(* Logix 5000 project; controller _2081 vendor 1 type 14 code 77 rev 19.11; software revision 19.01; part 3 of 4 *)
(* tags used below, declared in another part *)
   B10 : DINT[255];   // Product Shift Register
   B23 : DINT[20];   // Fault Bits
   B3 : DINT[10];   // Utility Bits
   B33 : DINT[10];   // Utility Bits
   B36 : DINT[10];   // One-Shots
   B37 : DINT[10];   // Product Location
   C5 : COUNTER[15];   // Line Duration Counters
   F38 : REAL[25];
   i3 : INT;   // Slot 3 16pt DC Input
   i4 : INT;   // Slot 4 16pt DC Input
   IR_1_BITOff : DINT;   // Indirect Addressing BIT Offset
   IR_1_DWOff : DINT;   // Indirect Addressing WORD Offset
   IR_BITOff : DINT;
   IR_DWOff : DINT;
   N26 : DINT[600];   // Write to PLC
   N27 : DINT[400];   // Read from PLC
   N28 : DINT[200];   // Read from PLC
   N32 : DINT[200];
   N32_1 : DINT;   // Recipe to Run Offset Value
   N32_2 : DINT;   // Recipe Copy Utility
   N32_3 : DINT;   // Recipe Copy Utility
   N40 : DINT[256];   // Recipe Shift
   N41 : DINT[256];   // Recipe Shift
   N42 : DINT[256];   // Recipe Shift
   N50 : DINT[2500];   // Stored Recipes
   o2 : INT[8];   // Slot 2 8-pt Analog Output
   Offset : DINT;
   R6 : CONTROL[10];
   S24 : INT;   // Index Register
   T34 : TIMER[30];   // Utility Timers
   T4 : TIMER[32];
(* BGK_OVEN, continued *)

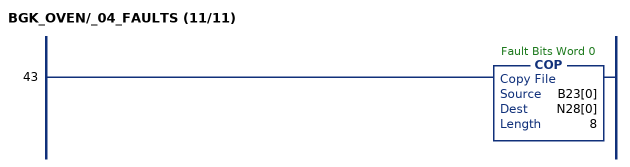
   [picture p24: BGK_OVEN/_04_FAULTS rungs 43-43]
   43: COP(B23[0],N28[0],8);
END_ROUTINE

ROUTINE _05_OIT_MAP   (* ladder *)
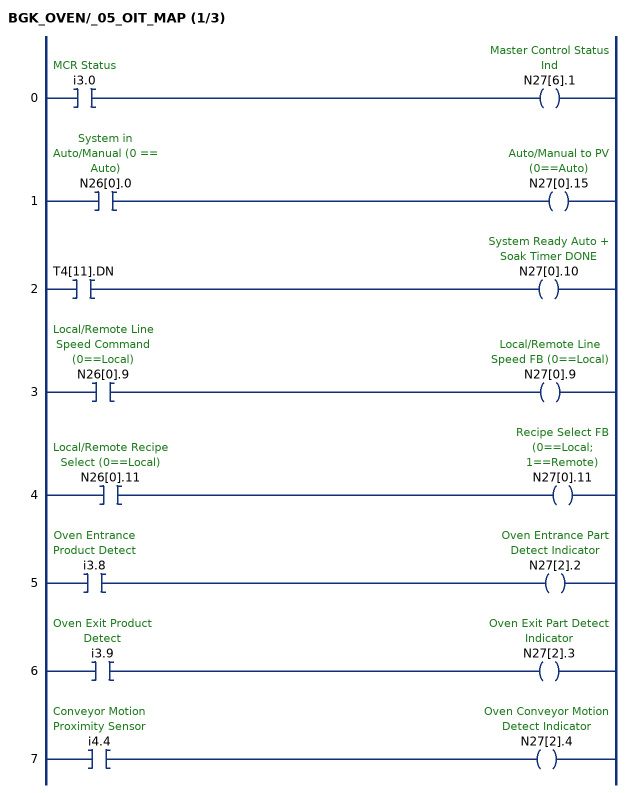
   0: XIC(i3.0)OTE(N27[6].1);
   1: XIC(N26[0].0)OTE(N27[0].15);
   2: XIC(T4[11].DN)OTE(N27[0].10);
   3: XIC(N26[0].9)OTE(N27[0].9);
   4: XIC(N26[0].11)OTE(N27[0].11);
   5: XIC(i3.8)OTE(N27[2].2);
   6: XIC(i3.9)OTE(N27[2].3);
   7: XIC(i4.4)OTE(N27[2].4);
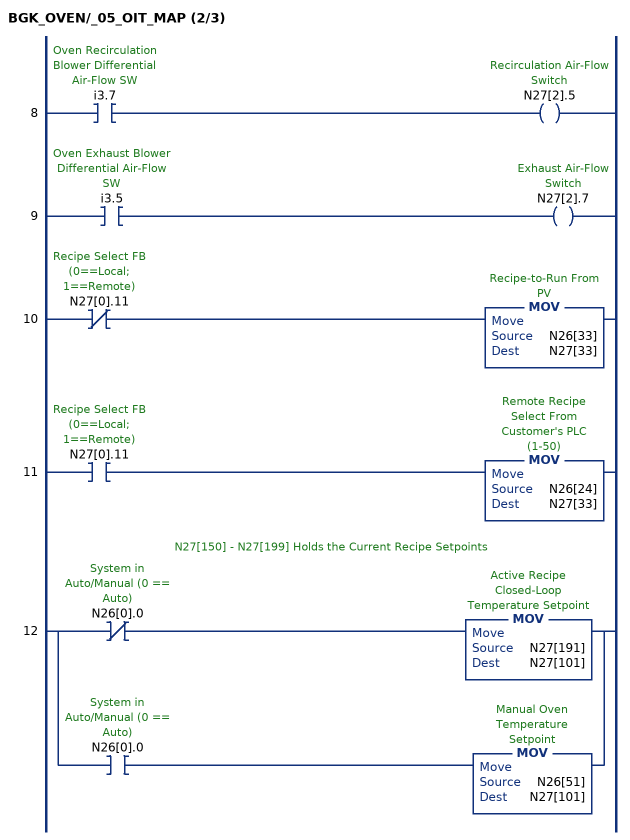
   8: XIC(i3.7)OTE(N27[2].5);
   9: XIC(i3.5)OTE(N27[2].7);
   10: XIO(N27[0].11)MOV(N26[33],N27[33]);
   11: XIC(N27[0].11)MOV(N26[24],N27[33]);
   // N27[150] - N27[199] Holds the Current Recipe Setpoints
   12: [XIO(N26[0].0) MOV(N27[191],N27[101]) ,XIC(N26[0].0) MOV(N26[51],N27[101]) ];
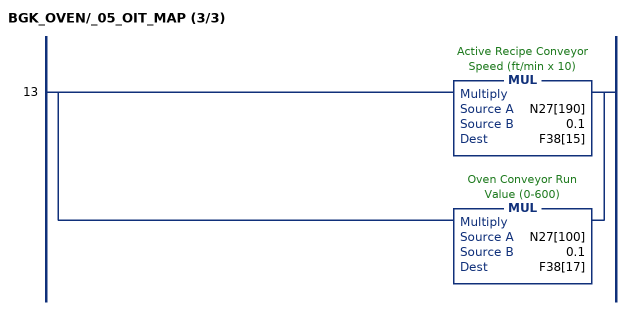
   13: [MUL(N27[190],0.1,F38[15]) ,MUL(N27[100],0.1,F38[17]) ];
END_ROUTINE

ROUTINE _06_SHIFT_REG   (* ladder *)
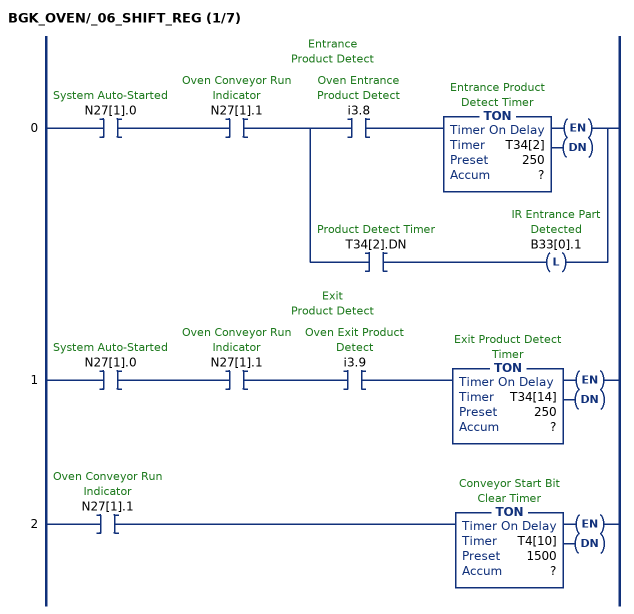
   // Entrance
   // Product Detect
   0: XIC(N27[1].0)XIC(N27[1].1)[XIC(i3.8) TON(T34[2],?,?) ,XIC(T34[2].DN) OTL(B33[0].1) ];
   // Exit
   // Product Detect
   1: XIC(N27[1].0)XIC(N27[1].1)XIC(i3.9)TON(T34[14],?,?);
   2: XIC(N27[1].1)TON(T4[10],?,?);
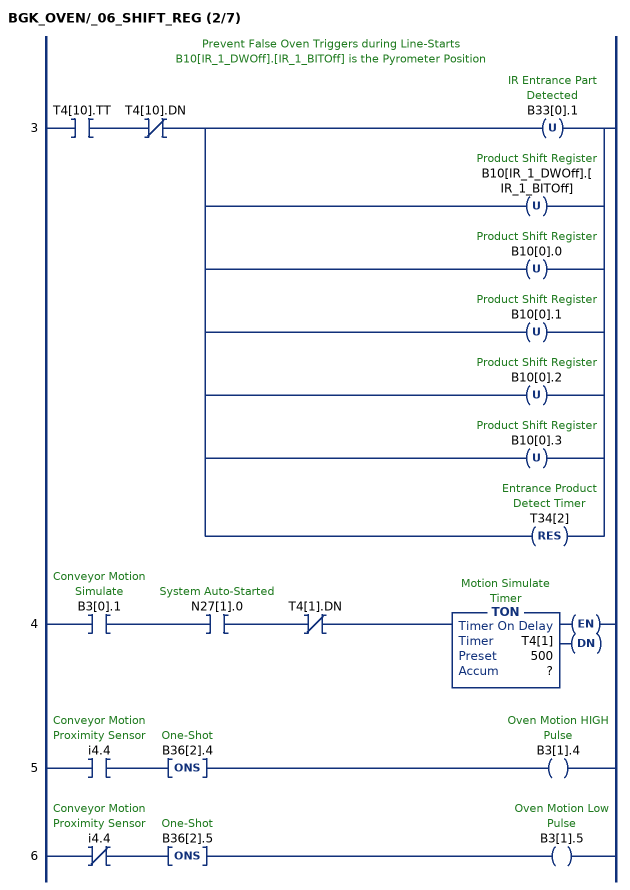
   // Prevent False Oven Triggers during Line-Starts
   // B10[IR_1_DWOff].[IR_1_BITOff] is the Pyrometer Position
   3: XIC(T4[10].TT)XIO(T4[10].DN)[OTU(B33[0].1) ,OTU(B10[IR_1_DWOff].[IR_1_BITOff]) ,OTU(B10[0].0) ,OTU(B10[0].1) ,OTU(B10[0].2) ,OTU(B10[0].3) ,RES(T34[2]) ];
   4: XIC(B3[0].1)XIC(N27[1].0)XIO(T4[1].DN)TON(T4[1],?,?);
   5: XIC(i4.4)ONS(B36[2].4)OTE(B3[1].4);
   6: XIO(i4.4)ONS(B36[2].5)OTE(B3[1].5);
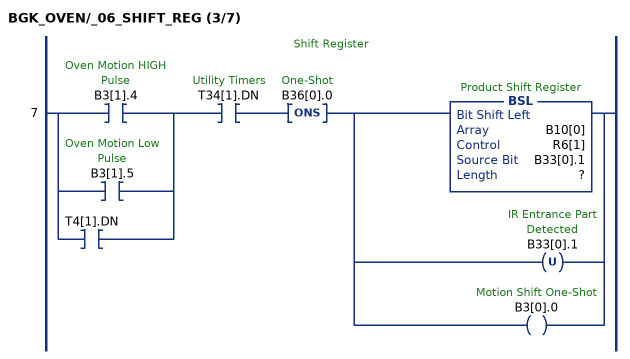
   // Shift Register
   7: [XIC(B3[1].4) ,XIC(B3[1].5) ,XIC(T4[1].DN) ]XIC(T34[1].DN)ONS(B36[0].0)[BSL(B10[0],R6[1],B33[0].1,?) ,OTU(B33[0].1) ,OTE(B3[0].0) ];
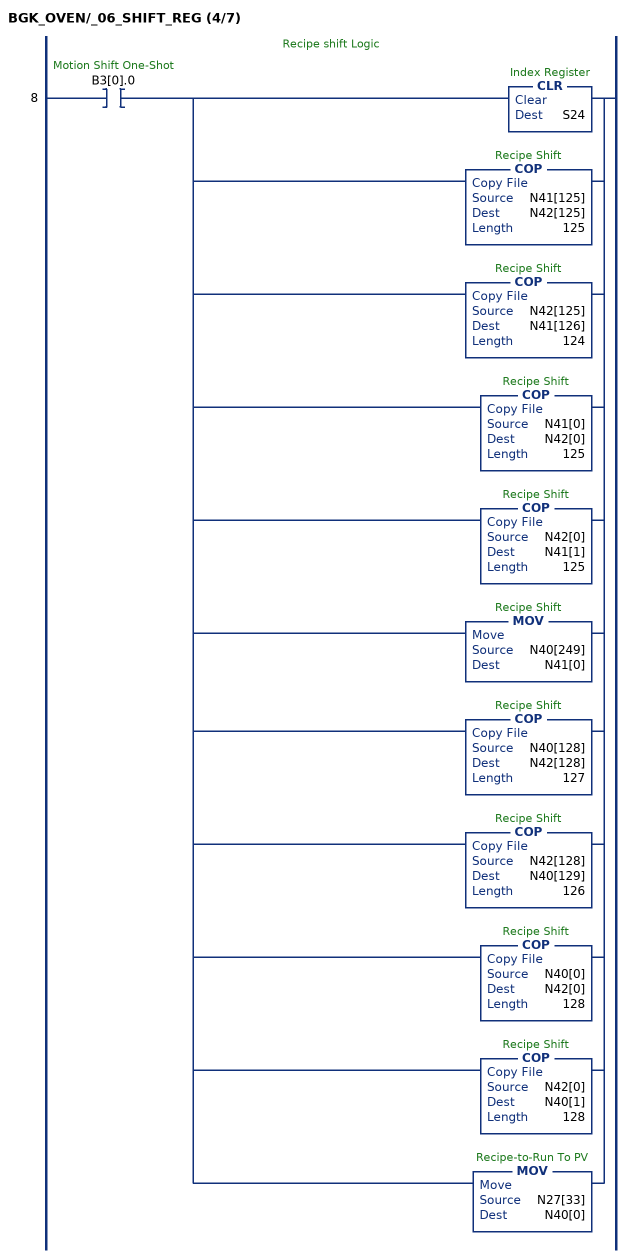
   // Recipe shift Logic
   8: XIC(B3[0].0)[CLR(S24) ,COP(N41[125],N42[125],125) ,COP(N42[125],N41[126],124) ,COP(N41[0],N42[0],125) ,COP(N42[0],N41[1],125) ,MOV(N40[249],N41[0]) ,COP(N40[128],N42[128],127) ,COP(N42[128],N40[129],126) ,COP(N40[0],N42[0],128) ,COP(N42[0],N40[1],128) ,MOV(N27[33],N40[0]) ];
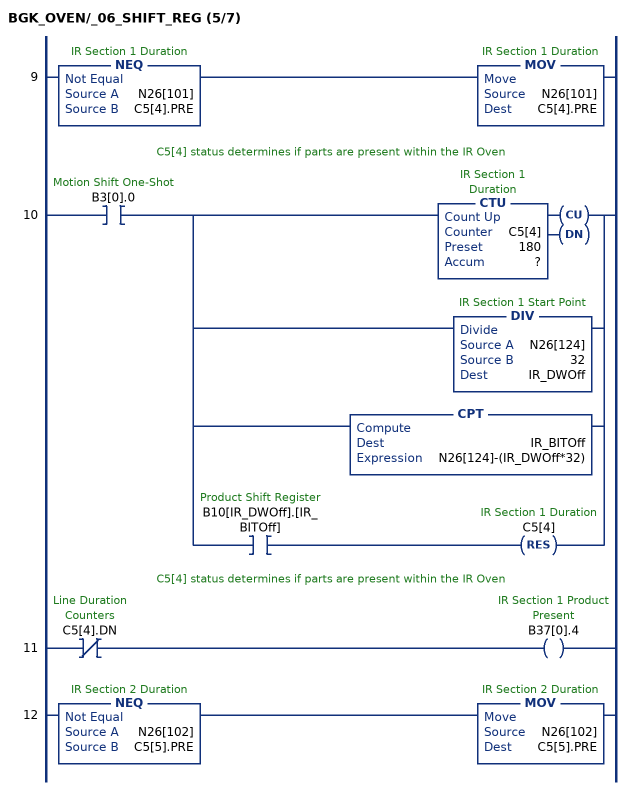
   9: NEQ(N26[101],C5[4].PRE)MOV(N26[101],C5[4].PRE);
   // C5[4] status determines if parts are present within the IR Oven
   10: XIC(B3[0].0)[CTU(C5[4],?,?) ,[DIV(N26[124],32,IR_DWOff) ,CPT(IR_BITOff,N26[124]-(IR_DWOff*32)) ] ,XIC(B10[IR_DWOff].[IR_BITOff]) RES(C5[4]) ];
   // C5[4] status determines if parts are present within the IR Oven
   11: XIO(C5[4].DN)OTE(B37[0].4);
   12: NEQ(N26[102],C5[5].PRE)MOV(N26[102],C5[5].PRE);
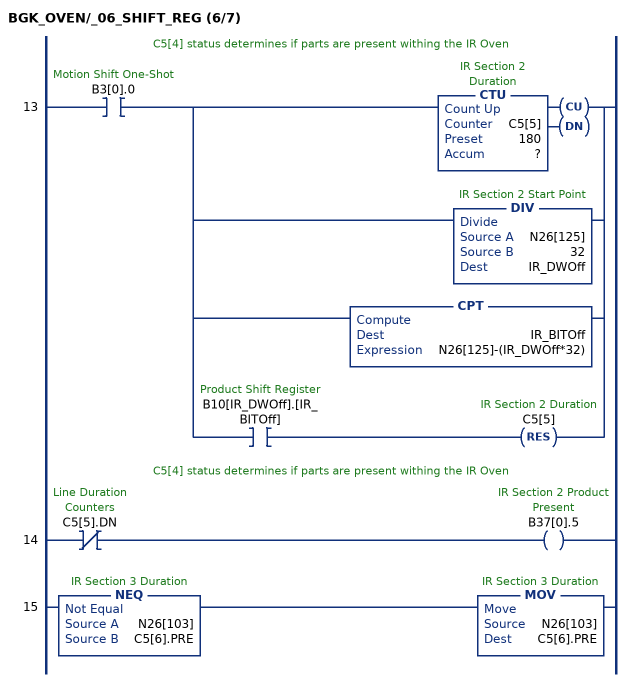
   // C5[4] status determines if parts are present withing the IR Oven
   13: XIC(B3[0].0)[CTU(C5[5],?,?) ,[DIV(N26[125],32,IR_DWOff) ,CPT(IR_BITOff,N26[125]-(IR_DWOff*32)) ] ,XIC(B10[IR_DWOff].[IR_BITOff]) RES(C5[5]) ];
   // C5[4] status determines if parts are present withing the IR Oven
   14: XIO(C5[5].DN)OTE(B37[0].5);
   15: NEQ(N26[103],C5[6].PRE)MOV(N26[103],C5[6].PRE);
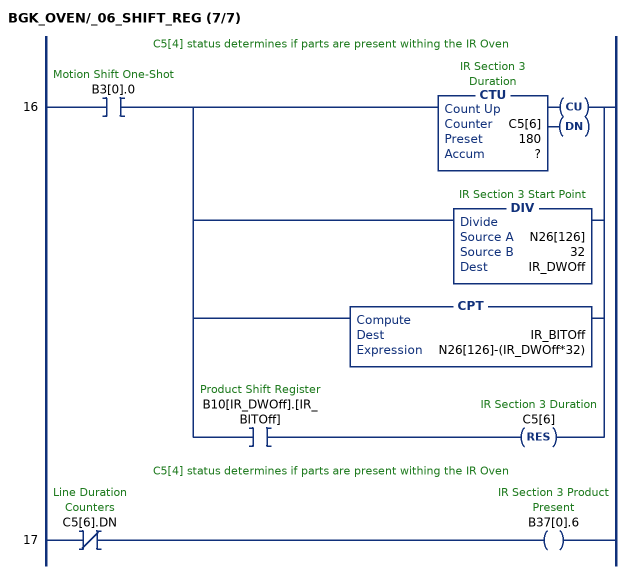
   // C5[4] status determines if parts are present withing the IR Oven
   16: XIC(B3[0].0)[CTU(C5[6],?,?) ,[DIV(N26[126],32,IR_DWOff) ,CPT(IR_BITOff,N26[126]-(IR_DWOff*32)) ] ,XIC(B10[IR_DWOff].[IR_BITOff]) RES(C5[6]) ];
   // C5[4] status determines if parts are present withing the IR Oven
   17: XIO(C5[6].DN)OTE(B37[0].6);
END_ROUTINE

ROUTINE _08_RECIPE   (* ladder *)
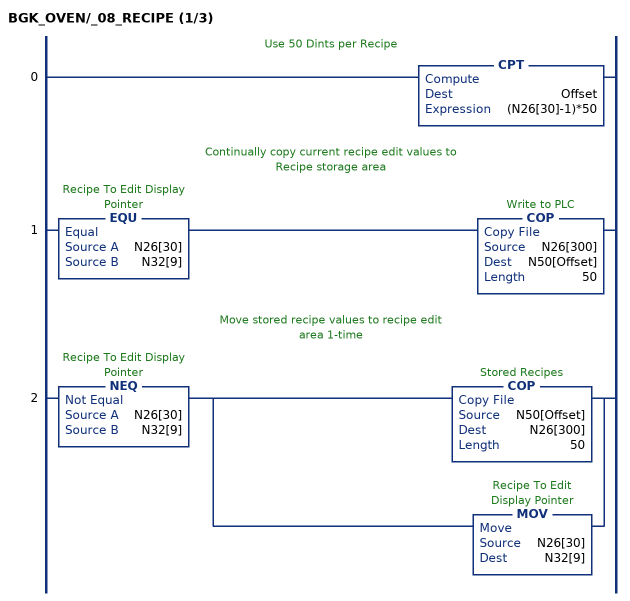
   // Use 50 Dints per Recipe
   0: CPT(Offset,(N26[30]-1)*50);
   // Continually copy current recipe edit values to
   // Recipe storage area
   1: EQU(N26[30],N32[9])COP(N26[300],N50[Offset],50);
   // Move stored recipe values to recipe edit
   // area 1-time
   2: NEQ(N26[30],N32[9])[COP(N50[Offset],N26[300],50) ,MOV(N26[30],N32[9]) ];
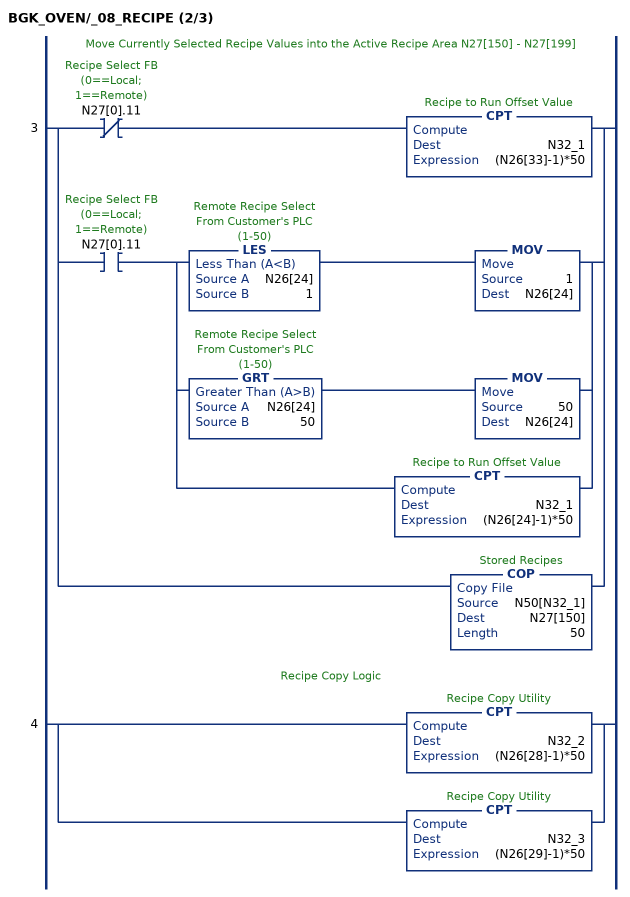
   // Move Currently Selected Recipe Values into the Active Recipe Area N27[150] - N27[199]
   3: [XIO(N27[0].11) CPT(N32_1,(N26[33]-1)*50) ,XIC(N27[0].11) [LES(N26[24],1) MOV(1,N26[24]) ,GRT(N26[24],50) MOV(50,N26[24]) ,CPT(N32_1,(N26[24]-1)*50) ] ,COP(N50[N32_1],N27[150],50) ];
   // Recipe Copy Logic
   4: [CPT(N32_2,(N26[28]-1)*50) ,CPT(N32_3,(N26[29]-1)*50) ];
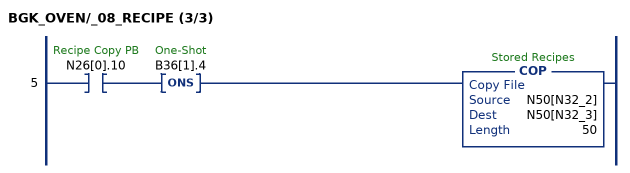
   5: XIC(N26[0].10)ONS(B36[1].4)COP(N50[N32_2],N50[N32_3],50);
END_ROUTINE

ROUTINE _11_ANALOG_OUT   (* ladder *)
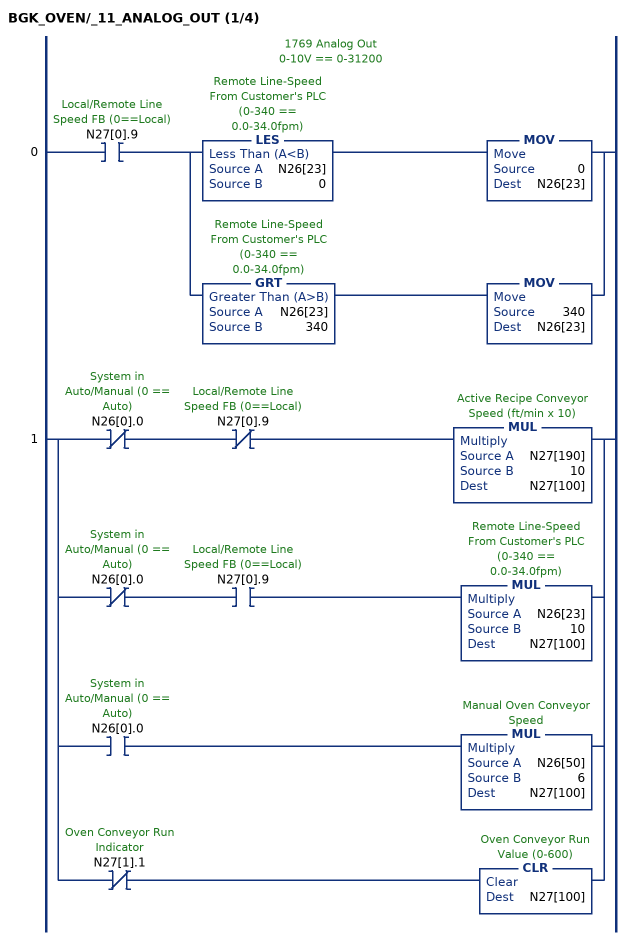
   // 1769 Analog Out
   // 0-10V == 0-31200
   0: XIC(N27[0].9)[LES(N26[23],0) MOV(0,N26[23]) ,GRT(N26[23],340) MOV(340,N26[23]) ];
   1: [XIO(N26[0].0) XIO(N27[0].9) MUL(N27[190],10,N27[100]) ,XIO(N26[0].0) XIC(N27[0].9) MUL(N26[23],10,N27[100]) ,XIC(N26[0].0) MUL(N26[50],6,N27[100]) ,XIO(N27[1].1) CLR(N27[100]) ];
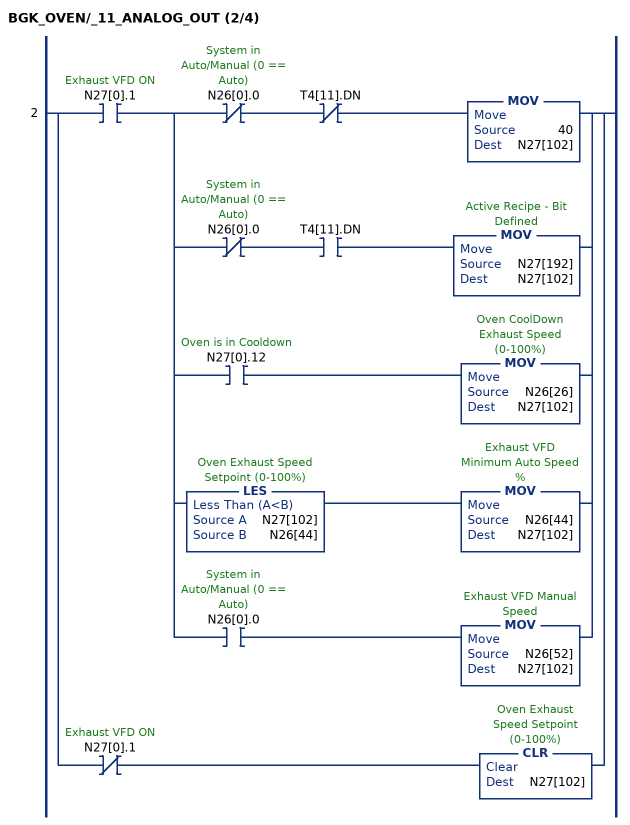
   2: [XIC(N27[0].1) [XIO(N26[0].0) XIO(T4[11].DN) MOV(40,N27[102]) ,XIO(N26[0].0) XIC(T4[11].DN) MOV(N27[192],N27[102]) ,XIC(N27[0].12) MOV(N26[26],N27[102]) ,LES(N27[102],N26[44]) MOV(N26[44],N27[102]) ,XIC(N26[0].0) MOV(N26[52],N27[102]) ] ,XIO(N27[0].1) CLR(N27[102]) ];
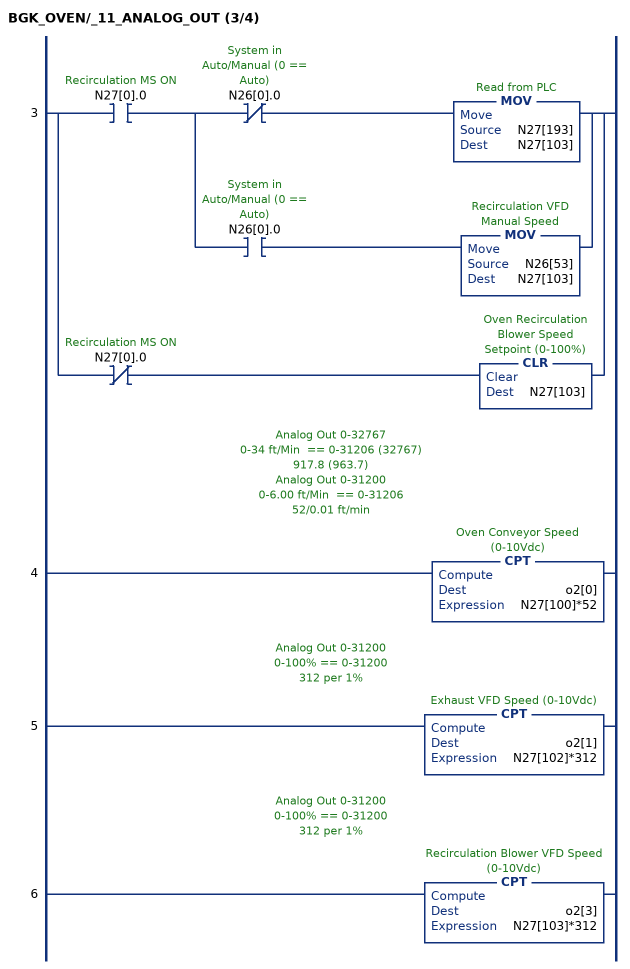
   3: [XIC(N27[0].0) [XIO(N26[0].0) MOV(N27[193],N27[103]) ,XIC(N26[0].0) MOV(N26[53],N27[103]) ] ,XIO(N27[0].0) CLR(N27[103]) ];
   // Analog Out 0-32767
   // 0-34 ft/Min  == 0-31206 (32767)
   // 917.8 (963.7)
   // Analog Out 0-31200
   // 0-6.00 ft/Min  == 0-31206
   // 52/0.01 ft/min
   4: CPT(o2[0],N27[100]*52);
   // Analog Out 0-31200
   // 0-100% == 0-31200
   // 312 per 1%
   5: CPT(o2[1],N27[102]*312);
   // Analog Out 0-31200
   // 0-100% == 0-31200
   // 312 per 1%
   6: CPT(o2[3],N27[103]*312);
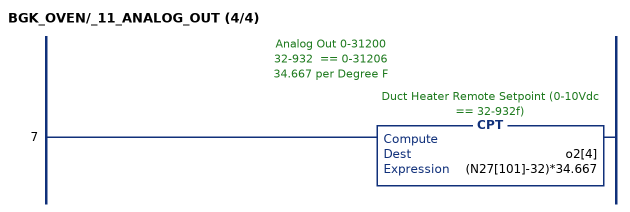
   // Analog Out 0-31200
   // 32-932  == 0-31206
   // 34.667 per Degree F
   7: CPT(o2[4],(N27[101]-32)*34.667);
END_ROUTINE
